// TIA Portal V18 export
VAR_GLOBAL   // PLC tag table "Cabinet_5_6"
   Sz5_ST01_SenA AT %I1504.0 : Bool;
   Sz5_ST01_SenB AT %I1504.1 : Bool;
   Sz5_ST01_SenC AT %I1504.2 : Bool;
   Sz5_ST01_SenD AT %I1504.3 : Bool;
   Sz5_ST02_SenA AT %I1504.4 : Bool;
   Sz5_ST02_SenB AT %I1504.5 : Bool;
   Sz5_ST02_SenC AT %I1504.6 : Bool;
   Sz5_ST02_SenD AT %I1504.7 : Bool;
   Sz5_ST34_SenA AT %I1505.0 : Bool;
   Sz5_ST34_SenB AT %I1505.1 : Bool;
   Sz5_ST34_SenC AT %I1505.2 : Bool;
   Sz5_ST34_SenD AT %I1505.3 : Bool;
   Sz5_ST35_SenA AT %I1505.4 : Bool;
   Sz5_ST35_SenB AT %I1505.5 : Bool;
   Sz5_ST35_SenC AT %I1505.6 : Bool;
   Sz5_ST35_SenD AT %I1505.7 : Bool;
   Sz5_ST38_SenA AT %I1506.0 : Bool;
   Sz5_ST38_SenB AT %I1506.1 : Bool;
   Sz5_ST38_SenC AT %I1506.2 : Bool;
   Sz5_ST38_SenD AT %I1506.3 : Bool;
END_VAR
